PROGRAM main
VAR
	Enable AT %QX0.0 : bool;
	DelayTimer : TOF;
	Output AT %QX0.1 : bool;
END_VAR

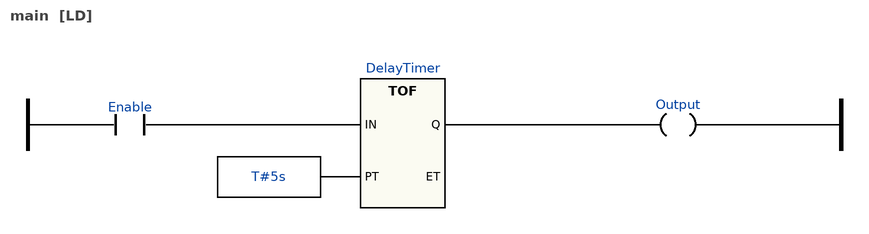
(* LD diagram, written out as Structured Text *)
DelayTimer(IN := Enable, PT := T#5s);
Output := DelayTimer.Q;
END_PROGRAM
